Universal Robots PolyScope program: main_ur_loop.urp

Program main_ur_loop (installation=default directory=/home/ur/ursim-current/programs createdIn=5.9.4.1031232 lastSavedIn=5.9.4.1031232 robotSerialNumber=20195599999)
Calibrated DH parameters: a=[0, -0.425, -0.3922, 0, 0, 0]; d=[0.1625, 0, 0, 0.1333, 0.0997, 0.0996]; alpha=[1.570796, 0, 0, 1.570796, -1.570796, 0]; deltaTheta=[0, 0, 0, 0, 0, 0]
BeforeStart
  socket1 := socket_open("192.168.0.7",8000)
  Script: movej([0,-3.1415/2, 3.1415/2, -3.1415/2, -3.1415/2, 0])
Robot Program (runOnlyOnce=false)
  Loop Forever
    Loop While (checkContinuously=false) expression=socket1≟False
      socket1 := socket_open("192.168.0.7",8000)
      Wait Sleep waitTime=0.5
    pose_position := get_actual_tcp_pose()
    Script: socket_send_string(pose_position)
    Wait Sleep waitTime=0.5
    jj := socket_read_ascii_float(5,timeout=0)
    Wait Sleep waitTime=0.5
    socket1 := False
    Script: socket_close()
    Script file /home/ur/ursim-current/programs/chess_movement_program.script
      | zlow = 0.05
      | zhigh = 0.4
      | 
      | pose1 = p[jj[2], jj[3], zlow, 3.1415, 0, 0]
      | pose2 = p[jj[2], jj[3], zhigh, 3.1415, 0, 0]
      | pose3 = p[jj[4], jj[5], zhigh, 3.1415, 0, 0]
      | pose4 = p[jj[4], jj[5], zlow, 3.1415, 0, 0]
      | 
      | if jj[1] == 1 :
      |   movel(pose3)
      |   sleep(2)
      |   movel(pose4)
      |   sleep(2)
      |   movel(pose3)
      |   sleep(1)
      | end
